Omron CX-Programmer project 新規ﾌﾟﾛｼﾞｪｸﾄ (CX-Programmer 9.61)

# PLC 新規PLC1: CP1L L

## Program 新規ﾌﾟﾛｸﾞﾗﾑ1 (cyclic task 0)

### Section ｾｸｼｮﾝ1

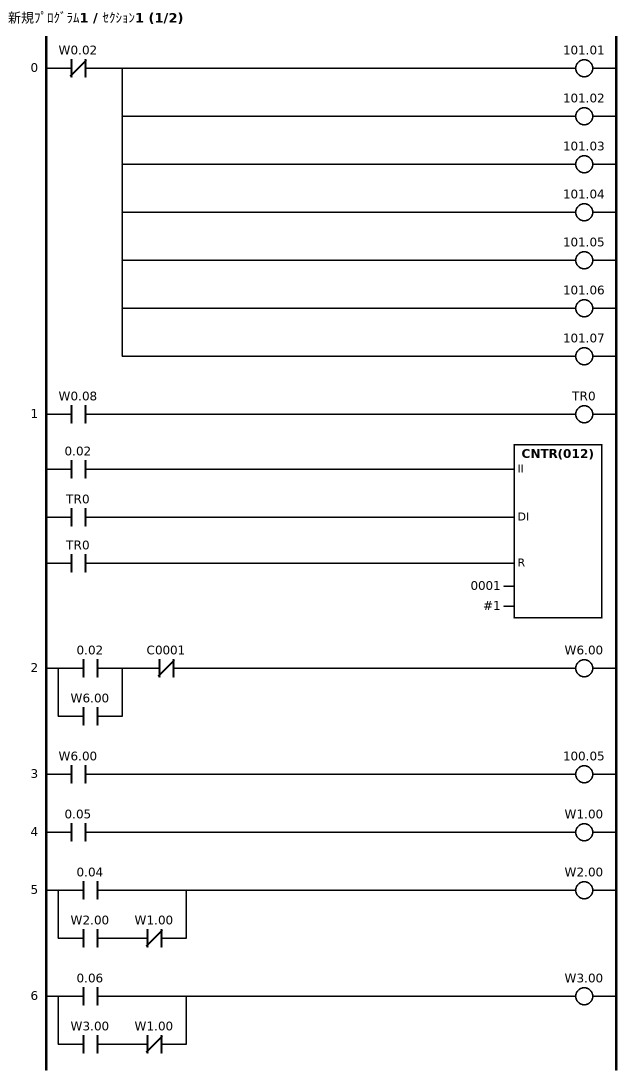
; rung 0
LDNOT W0.02
OUT 101.01
OUT 101.02
OUT 101.03
OUT 101.04
OUT 101.05
OUT 101.06
OUT 101.07
; rung 1
LD 0.02
LD W0.08
OUT TR0
LD TR0
CNTR(012) 0001 #1
; rung 2
LD 0.02
OR W6.00
ANDNOT C0001
OUT W6.00
; rung 3
LD W6.00
OUT 100.05
; rung 4
LD 0.05
OUT W1.00
; rung 5
LD 0.04
LD W2.00
ANDNOT W1.00
ORLD
OUT W2.00
; rung 6
LD 0.06
LD W3.00
ANDNOT W1.00
ORLD
OUT W3.00

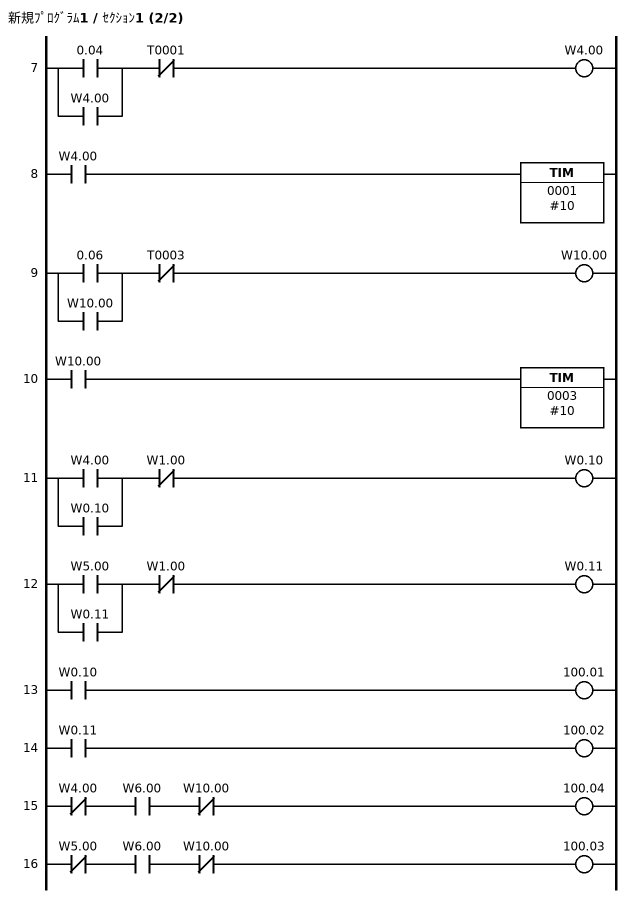
; rung 7
LD 0.04
OR W4.00
ANDNOT T0001
OUT W4.00
; rung 8
LD W4.00
TIM 0001 #10
; rung 9
LD 0.06
OR W10.00
ANDNOT T0003
OUT W10.00
; rung 10
LD W10.00
TIM 0003 #10
; rung 11
LD W4.00
OR W0.10
ANDNOT W1.00
OUT W0.10
; rung 12
LD W5.00
OR W0.11
ANDNOT W1.00
OUT W0.11
; rung 13
LD W0.10
OUT 100.01
; rung 14
LD W0.11
OUT 100.02
; rung 15
LDNOT W4.00
AND W6.00
ANDNOT W10.00
OUT 100.04
; rung 16
LDNOT W5.00
AND W6.00
ANDNOT W10.00
OUT 100.03

### Section END
; rung 0
END(001)